TYPE ST_ManualModeInputs :
STRUCT
    bSafetyOk                      : BOOL;
    bMotionSafetyPermitted         : BOOL;
    bTwoHandsSafe                  : BOOL;
    bProcessSafetyPermitted        : BOOL;
    bMainDoorSafe                  : BOOL;

    bIndexReady                    : BOOL;
    bIndexLocked                   : BOOL;
    bIndexBusy                     : BOOL;
    bIndexFaulted                  : BOOL;

    bSiliconeSupportExtended       : BOOL;
    bSiliconeSupportRetracted      : BOOL;
	bAssemblySupportExtended  	   : BOOL;
	bAssemblySupportRetracted 	   : BOOL;

    bProcessStationFaulted         : BOOL;

    bEquipmentReady                : BOOL;
    bEquipmentBusy                 : BOOL;
    bEquipmentFaulted              : BOOL;

    // Assembly / flipping station
    bAssemblyStationReady          : BOOL;
    bAssemblyStationBusy           : BOOL;
    bAssemblyStationFaulted        : BOOL;
    bAssemblyNestPartPresent       : BOOL;
    bAssemblyNestSiliconized       : BOOL;
    bAssemblyNestAlreadyAssembled  : BOOL;

    bReservoirPartPresent          : BOOL;

    // Manual Silicone Station
    bSiliconeProcessReady          : BOOL;
    bSiliconeProcessBusy           : BOOL;
    bSiliconeProcessFaulted        : BOOL;
    bSiliconeNestPartPresent       : BOOL;
    bSiliconeNestAlreadyProcessed  : BOOL;
	
	// IVEK Prime
	bIvekEnabled       			   : BOOL;
	bIvekFluidicReady 			   : BOOL;
	bIvekFluidicActive 			   : BOOL;
	bPartVacuumOk 					: BOOL;
	bIvekPrimeEnable 				: BOOL;
	bNozzlePressureOk              : BOOL;


END_STRUCT
END_TYPE

(* stored: Version 1.1.0.1, ProductVersion 3.1.4026.18
   DUT ST_ManualModeInputs: Id {18456921-6213-41f6-a504-07e7e56d014a} *)
